{attribute addProperty BoxType "EL3751-0000-0020"}
{attribute addProperty Id "PAI_StatusAT %I*PAI_Status_CF7232B03240PAI_Samples_1AT %I*PAI_Samples_4FE6FA0C3240PAI_TimestampAT %I*PAI_Timestamp_54B31DA16480WcStateAT %I*WcState_98A4DF7520.250InfoDataAT %I*InfoData_0BDED7BF144180"}
{attribute addProperty CRC "3557354704"}
{attribute addProperty SizeInBites "274"}
{attribute addProperty SizeInBytes "34.25"}
TYPE EL3751_1042CC80 :
STRUCT
	{attribute addProperty Name "PAI_Status"}
	PAI_Status : PAI_Status_CF7232B0;
	{attribute addProperty Name "PAI_Samples_1"}
	PAI_Samples_1 : PAI_Samples_4FE6FA0C;
	{attribute addProperty Name "PAI_Timestamp"}
	PAI_Timestamp : PAI_Timestamp_54B31DA1;
	{attribute addProperty Name "WcState"}
	WcState : WcState_98A4DF75;
	{attribute addProperty Name "InfoData"}
	InfoData : InfoData_0BDED7BF;
END_STRUCT
END_TYPE

(* stored: Version 1.2.0.0, ProductVersion 3.1.4024.9
   DUT EL3751_1042CC80: Id {7dfb6020-91dc-4c75-84c9-bf9c2421591f} *)
